// TIA Portal V17 export
// export: Created 2025-06-26T07:49:43.7421012Z, ExportSetting WithDefaults, DisplayName Totally Integrated Automation Portal, DisplayVersion V17 Update 8, DisplayName TIA Portal Openness, DisplayVersion V17 Update 8, DisplayName TIA Portal Version Control Interface, DisplayVersion V17, DisplayName STEP 7 Professional, DisplayVersion V17 Update 8, DisplayName STEP 7 Safety, DisplayVersion V17 Update 6, DisplayName WinCC Advanced, DisplayVersion V17 Update 8
FUNCTION_BLOCK "fbCPCPumpSim"   // FB51, FBD
TITLE = CPC pump simulator
{ S7_Optimized_Access := 'TRUE' }
AUTHOR : Heaten
VERSION : 0.1
// stored: AutoNumber true, IsIECCheckEnabled false, IsRetainMemResEnabled false, MemoryReserve 100, SetENOAutomatically false, UDAEnableTagReadback false
   VAR_INPUT
      bOn : Bool;
      fSuction : Real;   // [kPa]
      fMaxDeltaP : Real;   // [kPa]
      fMinDeltaP : Real;   // [kPa]
      fCycleTime : Real;
   END_VAR
   VAR_OUTPUT
      fDischarge : Real;   // [kPa]
   END_VAR
   VAR
      fDeltaP : Real;   // Pressure rise over the pump
      eOn : R_TRIG;
   END_VAR
BEGIN

REGION Network 1: Preset pressure to max at pump start
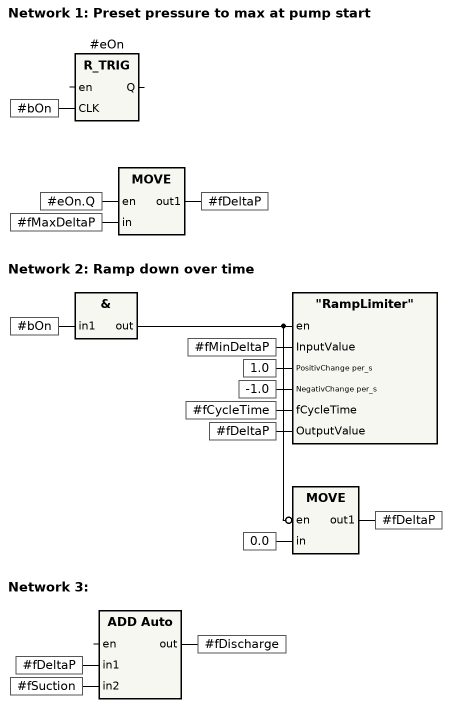
   #eOn(CLK := #bOn);   // R_TRIG
   IF #eOn.Q THEN #fDeltaP := #fMaxDeltaP; END_IF;
END_REGION

REGION Network 2: Ramp down over time
   // When pump is off, delta P is zero.
   // When the pump runs, it starts at the max pressure and ramps down to the min pressure to approximate the decrease in liquid on the suction side
   IF #bOn THEN
       "RampLimiter"(InputValue := #fMinDeltaP,
                     "PositivChange per_s" := 1.0,
                     "NegativChange per_s" := -1.0,
                     fCycleTime := #fCycleTime,
                     OutputValue := #fDeltaP);
   END_IF;
   IF NOT #bOn THEN #fDeltaP := 0.0; END_IF;
END_REGION

REGION Network 3
   #fDischarge := #fDeltaP + #fSuction;
END_REGION
END_FUNCTION_BLOCK
